(* Logix 5000 project; controller IF2_DEMO Emulate 5570 rev 20.12; software revision 20.04; part 3 of 8 *)
(* tags used below, declared in another part *)
   HMI_Motion : COUNTER;
   Next_Product : DINT;
   OEE_Part_Scrap_Old : DINT;
   OEE_Scrap_Labeler : DINT;
   OrderQty : DINT[4];
   PartCountRollOver : DINT;
   Product_Change : DINT;
   RefillLine : LineData;
   Timer1000ms : TIMER;
   Timer250ms : TIMER;
   WallClock : DINT[7];
   WC : WC[10];

PROGRAM FillerR   (* main routine MainRoutine *)
VAR
   Block_Delay : TIMER := (PRE := 15000);
   Blocked_L : BOOL;
   BottleNum : STRING;
   Ctrl_Bit : BOOL := 1;
   DownStream_Run : ALIAS FOR WC[3].EventTrigger[0].1;
   DownStream_Running : ALIAS FOR WC[3].EventTrigger[0].8;
   Events : Events := (DownTime.BreakdownCode := 6, Control.StandbyCode := 1, Control.Run := 1, Control.Auto := 1);
   Events_Control_Auto : ALIAS FOR WC_L.EventTrigger[0].5;
   Events_Control_OpStop : ALIAS FOR WC_L.EventTrigger[0].3;
   Events_Control_Run : ALIAS FOR WC_L.EventTrigger[0].1;
   Events_Control_Running : ALIAS FOR WC_L.EventTrigger[0].8;
   Events_Control_Standby : ALIAS FOR WC_L.EventTrigger[0].0;
   Events_Control_StandbyCode : ALIAS FOR WC_L.FlexREAL[1];
   Events_DownTime_Breakdown : ALIAS FOR WC_L.EventTrigger[0].2;
   Events_DownTime_BreakdownCode : ALIAS FOR WC_L.EventValue_REAL[2];
   Events_DownTime_Testing : ALIAS FOR WC_L.EventTrigger[0].7;
   Events_DownTime_UnschedMaint : ALIAS FOR WC_L.EventTrigger[0].6;
   Events_Operate_Load : ALIAS FOR WC_L.EventTrigger[0].10;
   Events_Operate_OrderProc : ALIAS FOR WC_L.EventTrigger[0].11;
   Events_Operate_Setup : ALIAS FOR WC_L.EventTrigger[0].9;
   FillOunces : INT;
   HMI : HMIVars := (ScrapRate := 5.0, SpeedControl := 100.0, PrevSpeed := 100.0, PartCountRollOver := 9999999, MfgTimeBase := 1, MaxEventDur := 14.0, MinEventDur := 5.0, EventsPerHr := 55, EventDur := 12.487433, RunDur := 51.79828, MinRunDur := 5.0);
   MfgOrders : MfgOrders := (CustomerName := 'Big-Mart', OrderName := 'BB21', OrderQty := 30000, ProdRate := 60.0, SetupTime := 37.0, PartName := 'STRAW-R40', WorkcellName := 'FillerR', OperationId := 17160304, PartNameSav := 'STRAW-R40');
   MfgOrders_CustomerName : ALIAS FOR WC_L.FlexSTRING[4];
   MfgOrders_OrderName : ALIAS FOR WC_L.FlexSTRING[3];
   MfgOrders_PartName : ALIAS FOR WC_L.FlexSTRING[0];
   Motion : DINT := 31;
   Motion_Counter : DINT := 2;
   Motion_Speed : DINT := 10;
   MotionCount : TIMER := (PRE := 900);
   OEE : OEE := (IdealCycleTime := 3.0);
   OEE_IdealCycleTime : ALIAS FOR WC_L.IdealCT;
   OEE_Parts_Good : ALIAS FOR WC_L.GoodParts;
   OEE_Parts_Scrap : ALIAS FOR WC_L.ScrapParts;
   OEE_Parts_Total : ALIAS FOR WC_L.TotalParts;
   onsbits : DINT;
   OperatorID : ALIAS FOR WC_L.FlexREAL[1];
   Pressure1 : ALIAS FOR WC_L.PV[0];   // PSI
   ProductColorCode : INT := 2;
   RecipeName : STRING;
   SIM : SimVars := (Run.PRE := 51798, Event.PRE := 5000, Setup.PRE := 5000, EventNumber := 11, UtilityBool[2] := 1);
        .UTILITYBOOL[2]   // First Scan Bit
   Starve_Delay : TIMER := (PRE := 15000);
   Starved_L : BOOL;
   StateValue : ALIAS FOR WC_L.MonitorValue[0];
   Suppress : Events;
   Temperature1 : ALIAS FOR WC_L.PV[1];   // DEG
   UpStream_Run : BOOL := 1;
   UpStream_Running : BOOL := 1;   // Not used-no upstream wc
   WC_L : ALIAS FOR WC[1];
END_VAR

ROUTINE MainRoutine   (* ladder *)
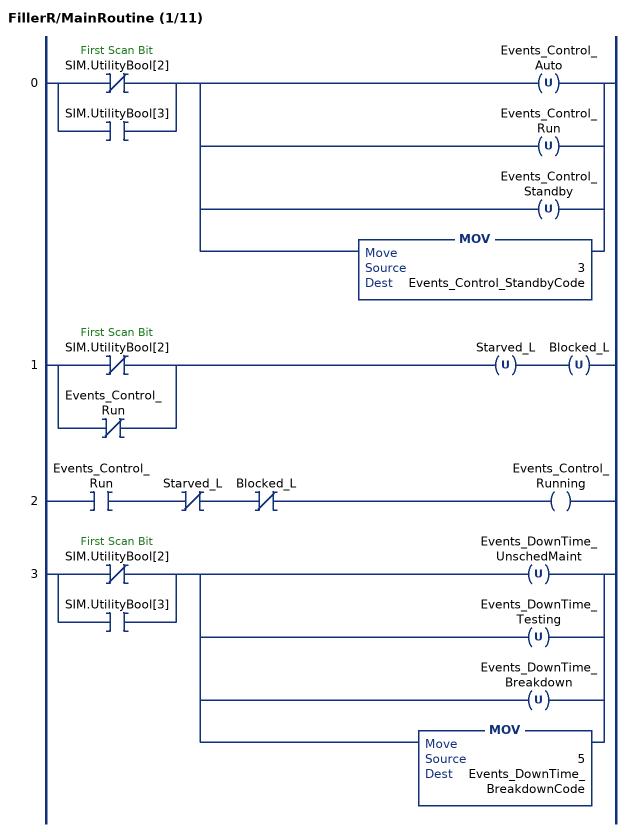
   0: [XIO(SIM.UtilityBool[2]) ,XIC(SIM.UtilityBool[3]) ][OTU(Events_Control_Auto) ,OTU(Events_Control_Run) ,OTU(Events_Control_Standby) ,MOV(3,Events_Control_StandbyCode) ];
   1: [XIO(SIM.UtilityBool[2]) ,XIO(Events_Control_Run) ]OTU(Starved_L)OTU(Blocked_L);
   2: XIC(Events_Control_Run)XIO(Starved_L)XIO(Blocked_L)OTE(Events_Control_Running);
   3: [XIO(SIM.UtilityBool[2]) ,XIC(SIM.UtilityBool[3]) ][OTU(Events_DownTime_UnschedMaint) ,OTU(Events_DownTime_Testing) ,OTU(Events_DownTime_Breakdown) ,MOV(5,Events_DownTime_BreakdownCode) ];
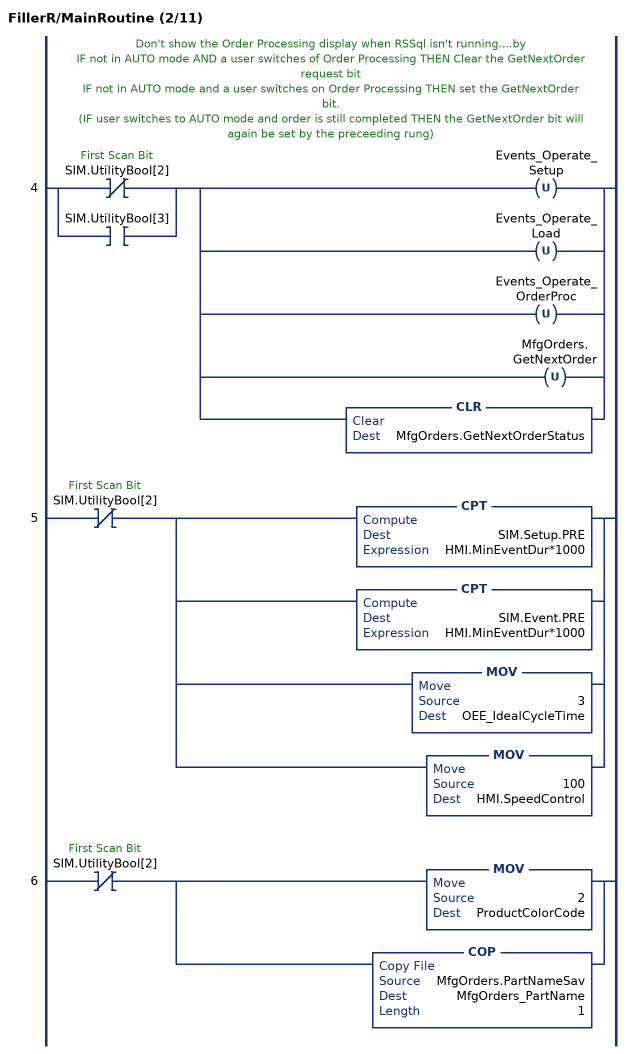
   // Don't show the Order Processing display when RSSql isn't running....by
   // IF not in AUTO mode AND a user switches of Order Processing THEN Clear the GetNextOrder request bit
   // IF not in AUTO mode and a user switches on Order Processing THEN set the GetNextOrder bit.
   // (IF user switches to AUTO mode and order is still completed THEN the GetNextOrder bit will again be set by the preceeding rung)
   4: [XIO(SIM.UtilityBool[2]) ,XIC(SIM.UtilityBool[3]) ][OTU(Events_Operate_Setup) ,OTU(Events_Operate_Load) ,OTU(Events_Operate_OrderProc) ,OTU(MfgOrders.GetNextOrder) ,CLR(MfgOrders.GetNextOrderStatus) ];
   5: XIO(SIM.UtilityBool[2])[CPT(SIM.Setup.PRE,HMI.MinEventDur*1000) ,CPT(SIM.Event.PRE,HMI.MinEventDur*1000) ,MOV(3,OEE_IdealCycleTime) ,MOV(100,HMI.SpeedControl) ];
   6: XIO(SIM.UtilityBool[2])[MOV(2,ProductColorCode) ,COP(MfgOrders.PartNameSav,MfgOrders_PartName,1) ];
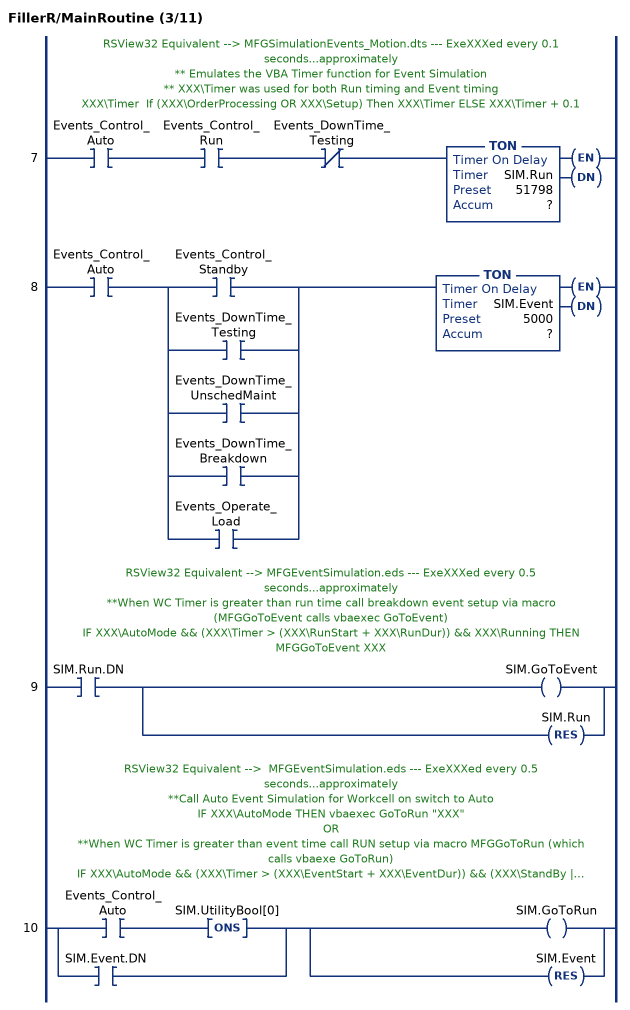
   // RSView32 Equivalent --> MFGSimulationEvents_Motion.dts --- ExeXXXed every 0.1 seconds...approximately
   // ** Emulates the VBA Timer function for Event Simulation
   // ** XXX\Timer was used for both Run timing and Event timing
   // XXX\Timer	If (XXX\OrderProcessing OR XXX\Setup) Then XXX\Timer ELSE XXX\Timer + 0.1
   7: XIC(Events_Control_Auto)XIC(Events_Control_Run)XIO(Events_DownTime_Testing)TON(SIM.Run,?,?);
   8: XIC(Events_Control_Auto)[XIC(Events_Control_Standby) ,XIC(Events_DownTime_Testing) ,XIC(Events_DownTime_UnschedMaint) ,XIC(Events_DownTime_Breakdown) ,XIC(Events_Operate_Load) ]TON(SIM.Event,?,?);
   // RSView32 Equivalent --> MFGEventSimulation.eds --- ExeXXXed every 0.5 seconds...approximately
   // **When WC Timer is greater than run time call breakdown event setup via macro (MFGGoToEvent calls vbaexec GoToEvent)
   // IF XXX\AutoMode && (XXX\Timer > (XXX\RunStart + XXX\RunDur)) && XXX\Running THEN MFGGoToEvent XXX
   9: XIC(SIM.Run.DN)[OTE(SIM.GoToEvent) ,RES(SIM.Run) ];
   // RSView32 Equivalent -->  MFGEventSimulation.eds --- ExeXXXed every 0.5 seconds...approximately
   // **Call Auto Event Simulation for Workcell on switch to Auto
   // IF XXX\AutoMode THEN vbaexec GoToRun "XXX"
   // OR
   // **When WC Timer is greater than event time call RUN setup via macro MFGGoToRun (which calls vbaexe GoToRun)
   // IF XXX\AutoMode && (XXX\Timer > (XXX\EventStart + XXX\EventDur)) && (XXX\StandBy || XXX\Test || XXX\UnSchedMaint || XXX\Breakdown ||XXX\Load) THEN MFGGoToRun XXX
   10: [XIC(Events_Control_Auto) ONS(SIM.UtilityBool[0]) ,XIC(SIM.Event.DN) ][OTE(SIM.GoToRun) ,RES(SIM.Event) ];
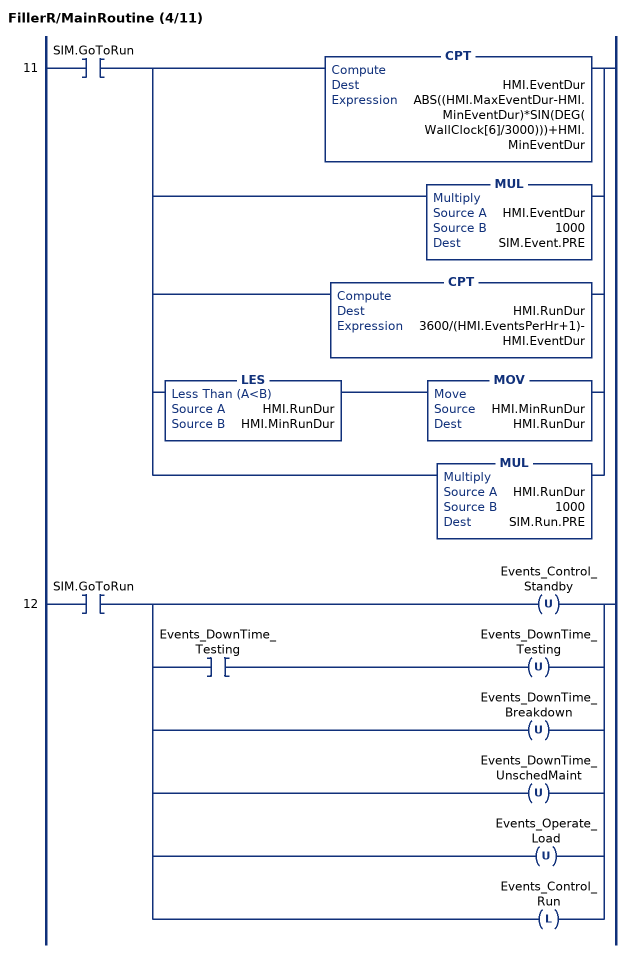
   11: XIC(SIM.GoToRun)[CPT(HMI.EventDur,ABS((HMI.MaxEventDur-HMI.MinEventDur)*SIN(DEG(WallClock[6]/3000)))+HMI.MinEventDur) ,MUL(HMI.EventDur,1000,SIM.Event.PRE) ,CPT(HMI.RunDur,3600/(HMI.EventsPerHr+1)-HMI.EventDur) ,LES(HMI.RunDur,HMI.MinRunDur) MOV(HMI.MinRunDur,HMI.RunDur) ,MUL(HMI.RunDur,1000,SIM.Run.PRE) ];
   12: XIC(SIM.GoToRun)[OTU(Events_Control_Standby) ,XIC(Events_DownTime_Testing) OTU(Events_DownTime_Testing) ,OTU(Events_DownTime_Breakdown) ,OTU(Events_DownTime_UnschedMaint) ,OTU(Events_Operate_Load) ,OTL(Events_Control_Run) ];
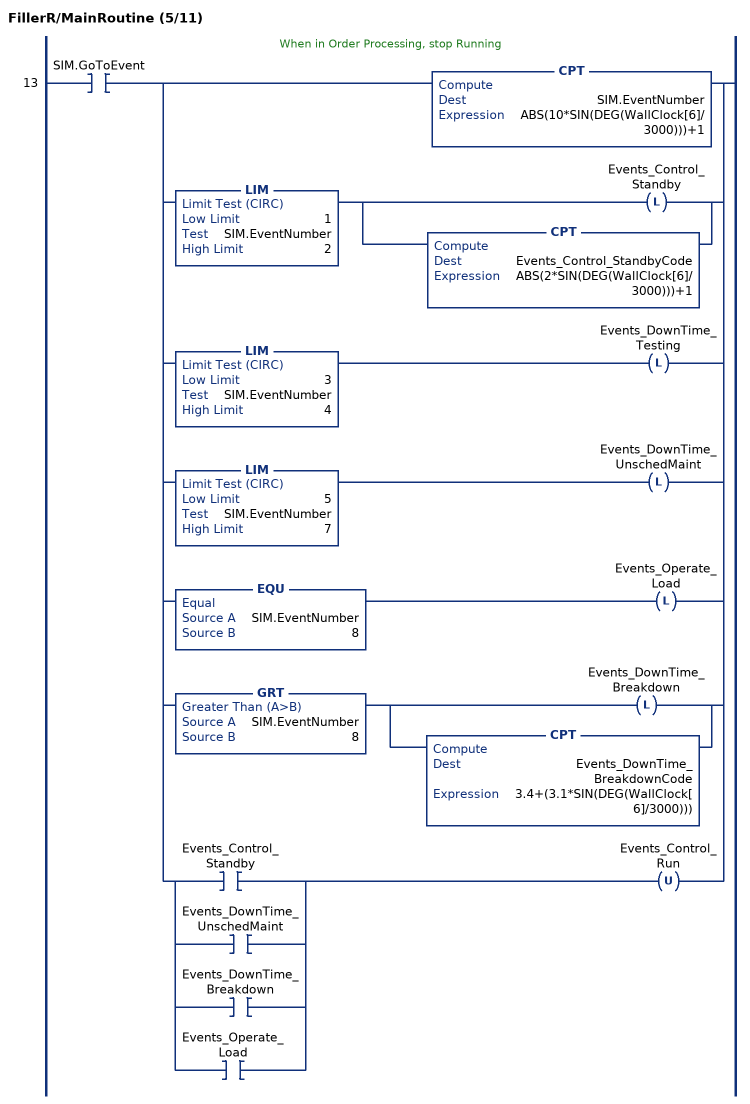
   // When in Order Processing, stop Running
   13: XIC(SIM.GoToEvent)[CPT(SIM.EventNumber,ABS(10*SIN(DEG(WallClock[6]/3000)))+1) ,LIM(1,SIM.EventNumber,2) [OTL(Events_Control_Standby) ,CPT(Events_Control_StandbyCode,ABS(2*SIN(DEG(WallClock[6]/3000)))+1) ] ,LIM(3,SIM.EventNumber,4) OTL(Events_DownTime_Testing) ,LIM(5,SIM.EventNumber,7) OTL(Events_DownTime_UnschedMaint) ,EQU(SIM.EventNumber,8) OTL(Events_Operate_Load) ,GRT(SIM.EventNumber,8) [OTL(Events_DownTime_Breakdown) ,CPT(Events_DownTime_BreakdownCode,3.4+(3.1*SIN(DEG(WallClock[6]/3000)))) ] ,[XIC(Events_Control_Standby) ,XIC(Events_DownTime_UnschedMaint) ,XIC(Events_DownTime_Breakdown) ,XIC(Events_Operate_Load) ] OTU(Events_Control_Run) ];
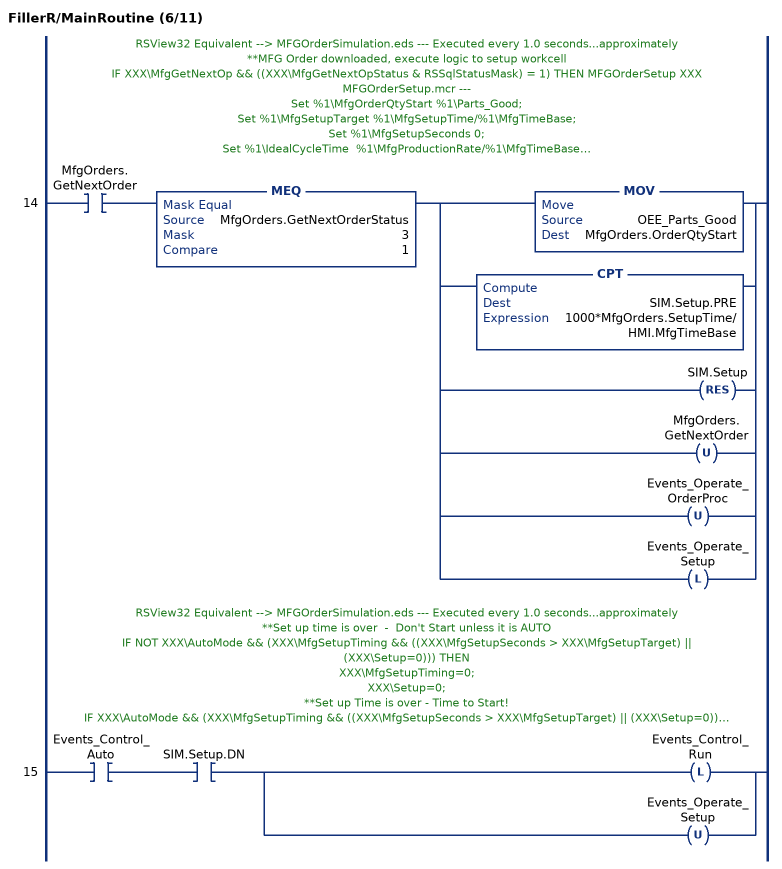
   // RSView32 Equivalent --> MFGOrderSimulation.eds --- Executed every 1.0 seconds...approximately
   // **MFG Order downloaded, execute logic to setup workcell
   // IF XXX\MfgGetNextOp && ((XXX\MfgGetNextOpStatus & RSSqlStatusMask) = 1) THEN MFGOrderSetup XXX
   // MFGOrderSetup.mcr ---
   // 	Set %1\MfgOrderQtyStart %1\Parts_Good;
   // 	Set %1\MfgSetupTarget %1\MfgSetupTime/%1\MfgTimeBase;
   // 	Set %1\MfgSetupSeconds 0;
   // 	Set %1\IdealCycleTime  %1\MfgProductionRate/%1\MfgTimeBase;
   // 	Set %1\MfgGetNextOp 0;
   // 	Set %1\Setup 1;
   // 	Set %1\OrderProcessing 0;
   // 	Set %1\MfgSetupTiming 1;
   14: XIC(MfgOrders.GetNextOrder)MEQ(MfgOrders.GetNextOrderStatus,3,1)[MOV(OEE_Parts_Good,MfgOrders.OrderQtyStart) ,CPT(SIM.Setup.PRE,1000*MfgOrders.SetupTime/HMI.MfgTimeBase) ,RES(SIM.Setup) ,OTU(MfgOrders.GetNextOrder) ,OTU(Events_Operate_OrderProc) ,OTL(Events_Operate_Setup) ];
   // RSView32 Equivalent --> MFGOrderSimulation.eds --- Executed every 1.0 seconds...approximately
   // **Set up time is over  -  Don't Start unless it is AUTO
   // IF NOT XXX\AutoMode && (XXX\MfgSetupTiming && ((XXX\MfgSetupSeconds > XXX\MfgSetupTarget) || (XXX\Setup=0))) THEN
   // 	XXX\MfgSetupTiming=0;
   // 	XXX\Setup=0;
   // **Set up Time is over - Time to Start!
   // IF XXX\AutoMode && (XXX\MfgSetupTiming && ((XXX\MfgSetupSeconds > XXX\MfgSetupTarget) || (XXX\Setup=0))) THEN
   // 	XXX\MfgSetupTiming=0;
   // 	XXX\Setup=0;
   // 	XXX\RUNNING=1
   15: XIC(Events_Control_Auto)XIC(SIM.Setup.DN)[OTL(Events_Control_Run) ,OTU(Events_Operate_Setup) ];
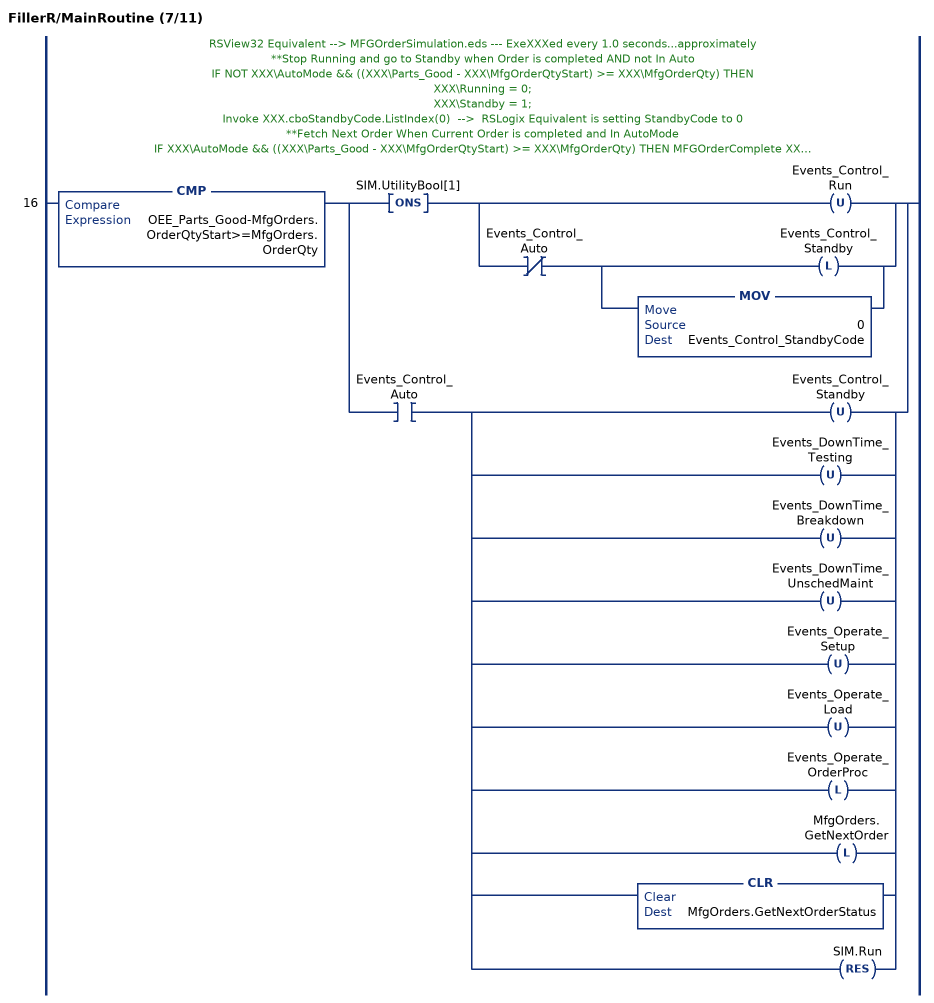
   // RSView32 Equivalent --> MFGOrderSimulation.eds --- ExeXXXed every 1.0 seconds...approximately
   // **Stop Running and go to Standby when Order is completed AND not In Auto
   // IF NOT XXX\AutoMode && ((XXX\Parts_Good - XXX\MfgOrderQtyStart) >= XXX\MfgOrderQty) THEN
   // 	XXX\Running = 0;
   // 	XXX\Standby = 1;
   // 	Invoke XXX.cboStandbyCode.ListIndex(0)  -->  RSLogix Equivalent is setting StandbyCode to 0
   // **Fetch Next Order When Current Order is completed and In AutoMode
   // IF XXX\AutoMode && ((XXX\Parts_Good - XXX\MfgOrderQtyStart) >= XXX\MfgOrderQty) THEN MFGOrderComplete XXX
   // MFGOrderComplete.mcr --- (Macros exeXXXed when called. %1 is the Workcell name -- typical all mcrs)
   // 	Set %1\RunStart %1\Timer;
   // 	Set %1\StandBy 0;
   // 	Set %1\Test 0;
   // 	Set %1\UnSchedMaint 0;
   // 	Set %1\Breakdown 0;
   // 	Set %1\Load 0;
   // 	Set %1\OrderProcessing 1;
   // 	Set %1\Running 0;
   // 	Set %1\MFGGetNextOpStatus 0;
   // 	Set %1\MFGGetNextOp 1
   16: CMP(OEE_Parts_Good-MfgOrders.OrderQtyStart>=MfgOrders.OrderQty)[ONS(SIM.UtilityBool[1]) [OTU(Events_Control_Run) ,XIO(Events_Control_Auto) [OTL(Events_Control_Standby) ,MOV(0,Events_Control_StandbyCode) ] ] ,XIC(Events_Control_Auto) [OTU(Events_Control_Standby) ,OTU(Events_DownTime_Testing) ,OTU(Events_DownTime_Breakdown) ,OTU(Events_DownTime_UnschedMaint) ,OTU(Events_Operate_Setup) ,OTU(Events_Operate_Load) ,OTL(Events_Operate_OrderProc) ,OTL(MfgOrders.GetNextOrder) ,CLR(MfgOrders.GetNextOrderStatus) ,RES(SIM.Run) ] ];
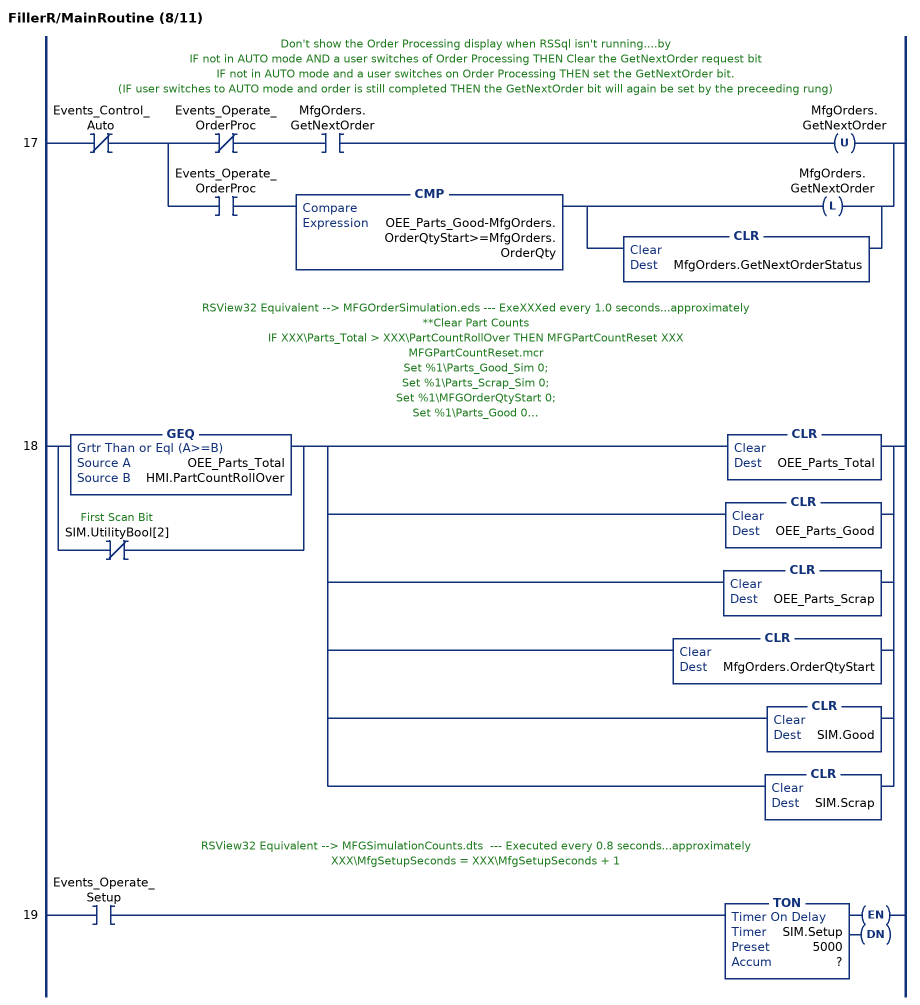
   // Don't show the Order Processing display when RSSql isn't running....by
   // IF not in AUTO mode AND a user switches of Order Processing THEN Clear the GetNextOrder request bit
   // IF not in AUTO mode and a user switches on Order Processing THEN set the GetNextOrder bit.
   // (IF user switches to AUTO mode and order is still completed THEN the GetNextOrder bit will again be set by the preceeding rung)
   17: XIO(Events_Control_Auto)[XIO(Events_Operate_OrderProc) XIC(MfgOrders.GetNextOrder) OTU(MfgOrders.GetNextOrder) ,XIC(Events_Operate_OrderProc) CMP(OEE_Parts_Good-MfgOrders.OrderQtyStart>=MfgOrders.OrderQty) [OTL(MfgOrders.GetNextOrder) ,CLR(MfgOrders.GetNextOrderStatus) ] ];
   // RSView32 Equivalent --> MFGOrderSimulation.eds --- ExeXXXed every 1.0 seconds...approximately
   // **Clear Part Counts
   // IF XXX\Parts_Total > XXX\PartCountRollOver THEN MFGPartCountReset XXX
   // MFGPartCountReset.mcr
   // 	Set %1\Parts_Good_Sim 0;
   // 	Set %1\Parts_Scrap_Sim 0;
   // 	Set %1\MFGOrderQtyStart 0;
   // 	Set %1\Parts_Good 0;
   // 	Set %1\Parts_Scrap 0;
   // 	Set %1\Parts_Total 0
   18: [GEQ(OEE_Parts_Total,HMI.PartCountRollOver) ,XIO(SIM.UtilityBool[2]) ][CLR(OEE_Parts_Total) ,CLR(OEE_Parts_Good) ,CLR(OEE_Parts_Scrap) ,CLR(MfgOrders.OrderQtyStart) ,CLR(SIM.Good) ,CLR(SIM.Scrap) ];
   // RSView32 Equivalent --> MFGSimulationCounts.dts	--- Executed every 0.8 seconds...approximately
   // XXX\MfgSetupSeconds = XXX\MfgSetupSeconds + 1
   19: XIC(Events_Operate_Setup)TON(SIM.Setup,?,?);
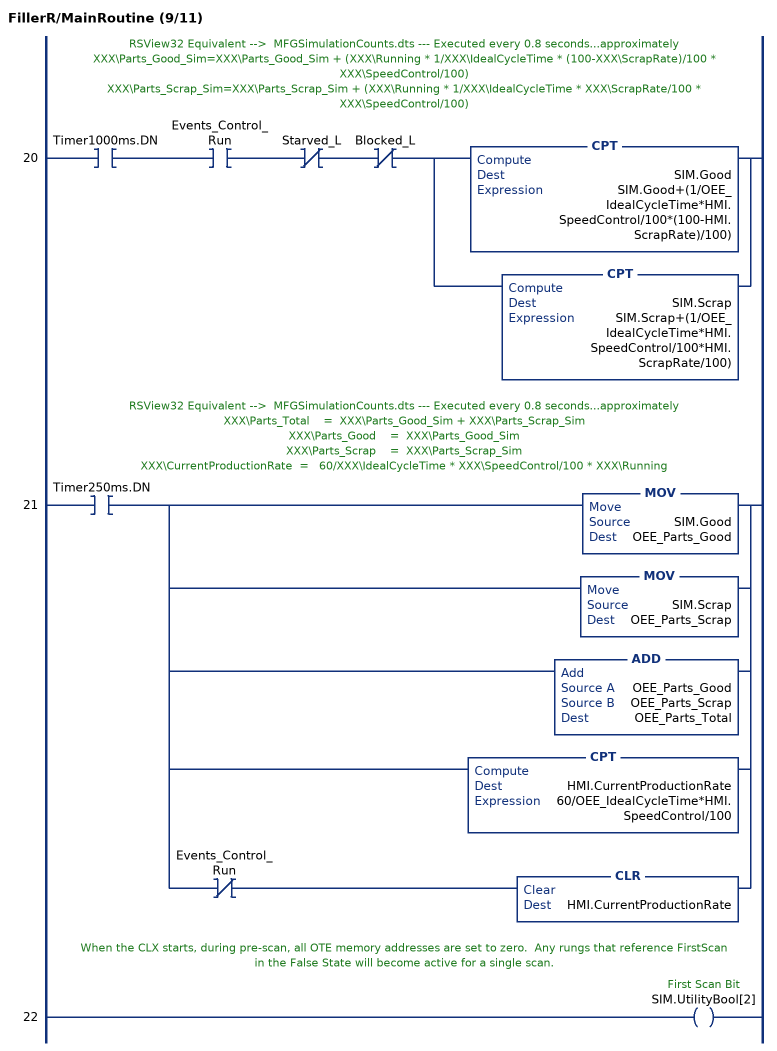
   // RSView32 Equivalent -->  MFGSimulationCounts.dts --- Executed every 0.8 seconds...approximately
   // XXX\Parts_Good_Sim=XXX\Parts_Good_Sim + (XXX\Running * 1/XXX\IdealCycleTime * (100-XXX\ScrapRate)/100 * XXX\SpeedControl/100)
   // XXX\Parts_Scrap_Sim=XXX\Parts_Scrap_Sim + (XXX\Running * 1/XXX\IdealCycleTime * XXX\ScrapRate/100 * XXX\SpeedControl/100)
   20: XIC(Timer1000ms.DN)XIC(Events_Control_Run)XIO(Starved_L)XIO(Blocked_L)[CPT(SIM.Good,SIM.Good+(1/OEE_IdealCycleTime*HMI.SpeedControl/100*(100-HMI.ScrapRate)/100)) ,CPT(SIM.Scrap,SIM.Scrap+(1/OEE_IdealCycleTime*HMI.SpeedControl/100*HMI.ScrapRate/100)) ];
   // RSView32 Equivalent -->  MFGSimulationCounts.dts --- Executed every 0.8 seconds...approximately
   // XXX\Parts_Total		=	XXX\Parts_Good_Sim + XXX\Parts_Scrap_Sim
   // XXX\Parts_Good		=	XXX\Parts_Good_Sim
   // XXX\Parts_Scrap		=	XXX\Parts_Scrap_Sim
   // XXX\CurrentProductionRate  = 	60/XXX\IdealCycleTime * XXX\SpeedControl/100 * XXX\Running
   21: XIC(Timer250ms.DN)[[MOV(SIM.Good,OEE_Parts_Good) ,MOV(SIM.Scrap,OEE_Parts_Scrap) ,ADD(OEE_Parts_Good,OEE_Parts_Scrap,OEE_Parts_Total) ] ,CPT(HMI.CurrentProductionRate,60/OEE_IdealCycleTime*HMI.SpeedControl/100) ,XIO(Events_Control_Run) CLR(HMI.CurrentProductionRate) ];
   // When the CLX starts, during pre-scan, all OTE memory addresses are set to zero.  Any rungs that reference FirstScan in the False State will become active for a single scan.
   22: OTE(SIM.UtilityBool[2]);
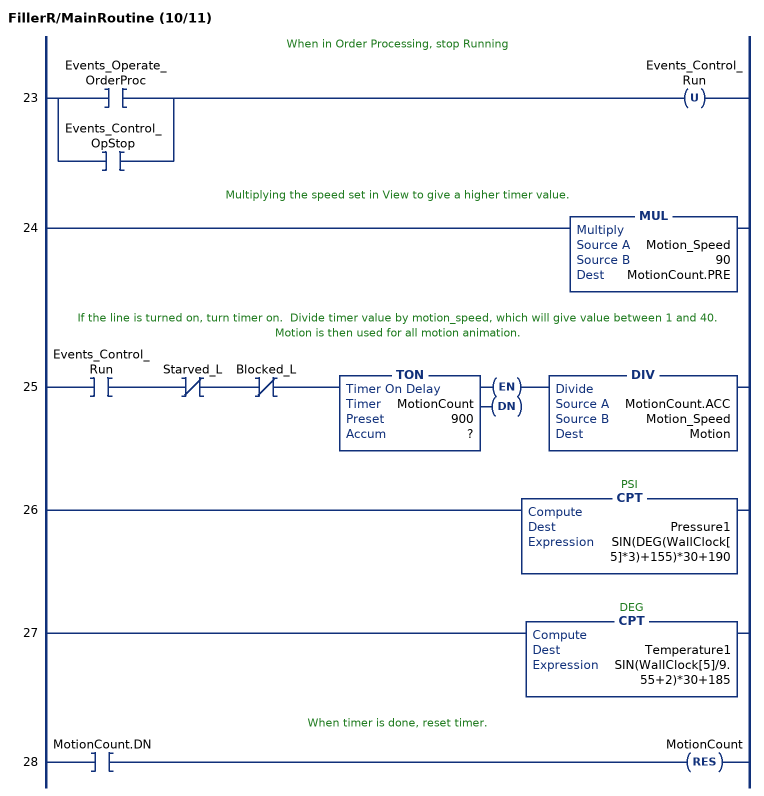
   // When in Order Processing, stop Running
   23: [XIC(Events_Operate_OrderProc) ,XIC(Events_Control_OpStop) ]OTU(Events_Control_Run);
   // Multiplying the speed set in View to give a higher timer value.
   24: MUL(Motion_Speed,90,MotionCount.PRE);
   // If the line is turned on, turn timer on.  Divide timer value by motion_speed, which will give value between 1 and 40.  Motion is then used for all motion animation.
   25: XIC(Events_Control_Run)XIO(Starved_L)XIO(Blocked_L)TON(MotionCount,?,?)DIV(MotionCount.ACC,Motion_Speed,Motion);
   26: CPT(Pressure1,SIN(DEG(WallClock[5]*3)+155)*30+190);
   27: CPT(Temperature1,SIN(WallClock[5]/9.55+2)*30+185);
   // When timer is done, reset timer.
   28: XIC(MotionCount.DN)RES(MotionCount);
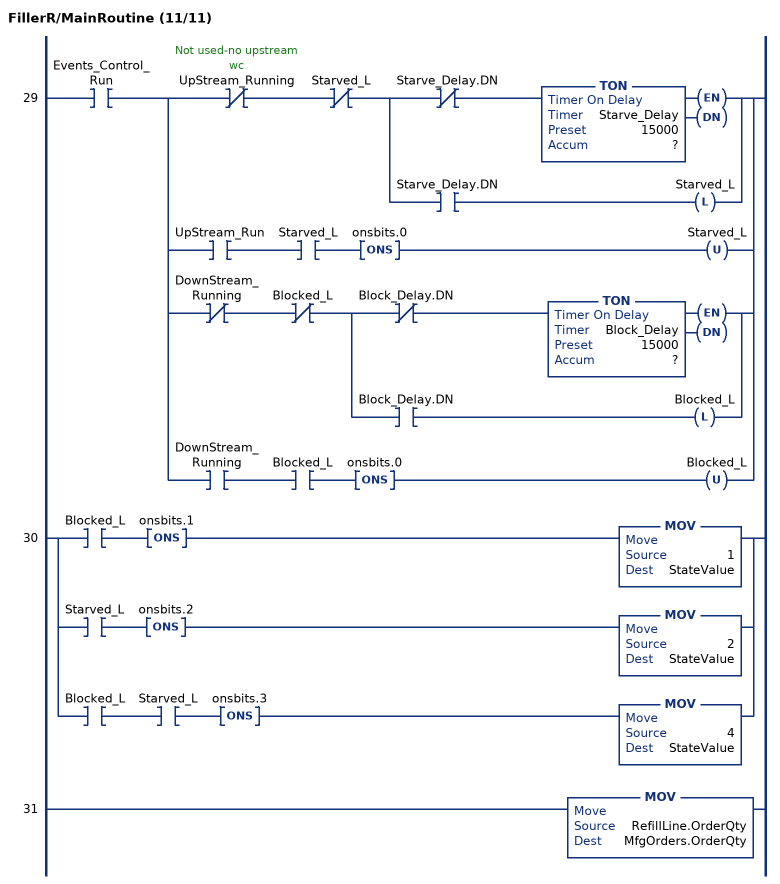
   29: XIC(Events_Control_Run)[[XIO(UpStream_Running) XIO(Starved_L) [XIO(Starve_Delay.DN) TON(Starve_Delay,?,?) ,XIC(Starve_Delay.DN) OTL(Starved_L) ] ,XIC(UpStream_Run) XIC(Starved_L) ONS(onsbits.0) OTU(Starved_L) ] ,[XIO(DownStream_Running) XIO(Blocked_L) [XIO(Block_Delay.DN) TON(Block_Delay,?,?) ,XIC(Block_Delay.DN) OTL(Blocked_L) ] ,XIC(DownStream_Running) XIC(Blocked_L) ONS(onsbits.0) OTU(Blocked_L) ] ];
   30: [XIC(Blocked_L) ONS(onsbits.1) MOV(1,StateValue) ,XIC(Starved_L) ONS(onsbits.2) MOV(2,StateValue) ,XIC(Blocked_L) XIC(Starved_L) ONS(onsbits.3) MOV(4,StateValue) ];
   31: MOV(RefillLine.OrderQty,MfgOrders.OrderQty);
END_ROUTINE
END_PROGRAM

PROGRAM LabelerD   (* main routine MainRoutine *)
VAR
   Alarm_Labeler1_Blocked : ALARM_DIGITAL;
   Alarm_Labeler1_Breakdown : ALARM_DIGITAL;
   Alarm_Labeler1_Starved : ALARM_DIGITAL;
   Alarm_Labeler1_Stopped : ALARM_DIGITAL;
   Block_Delay : TIMER := (PRE := 15000);
   Blocked_Condition : BOOL;
   Blocked_L : BOOL;
   BottleNum : STRING;
   Breakdown_Event_ONS : BOOL := 1;
   Breakdown_Labeler_Simulation : TIMER := (PRE := 300000, ACC := 53438, EN := 1, TT := 1);
   Breakdown_Labeler_Simulator_Down_Switch : BOOL;
   Breakdown_Occurance_Time : DINT := 260000;
   Breakdown_Variation_Stepper : DINT := 2;
   Ctrl_Bit : BOOL;
   DownStream_Run : ALIAS FOR WC[8].EventTrigger[0].1;
   DownStream_Running : ALIAS FOR WC[8].EventTrigger[0].8;
   Events : Events := (DownTime.BreakdownCode := 5, Control.StandbyCode := 1, Control.Run := 1, Control.Auto := 1);
   Events_Control_Auto : ALIAS FOR WC_L.EventTrigger[0].5;
   Events_Control_OpStop : ALIAS FOR WC_L.EventTrigger[0].3;
   Events_Control_Run : ALIAS FOR WC_L.EventTrigger[0].1;
   Events_Control_Running : ALIAS FOR WC_L.EventTrigger[0].8;
   Events_Control_Standby : ALIAS FOR WC_L.EventTrigger[0].0;
   Events_Control_StandbyCode : ALIAS FOR WC_L.EventValue_REAL[1];
   Events_DownTime_Breakdown : ALIAS FOR WC_L.EventTrigger[0].2;
   Events_DownTime_BreakdownCode : ALIAS FOR WC_L.EventValue_REAL[2];
   Events_DownTime_Testing : ALIAS FOR WC_L.EventTrigger[0].7;
   Events_DownTime_UnschedMaint : ALIAS FOR WC_L.EventTrigger[0].6;
   Events_Operate_Load : ALIAS FOR WC_L.EventTrigger[0].10;
   Events_Operate_OrderProc : ALIAS FOR WC_L.EventTrigger[0].11;
   Events_Operate_Setup : ALIAS FOR WC_L.EventTrigger[0].9;
   Expected_Full_Production_Rate : DINT := 113;
   FillOunces : INT;
   HMI : HMIVars := (ScrapRate := 6.0, SpeedControl := 400.0, PrevSpeed := 400.0, CurrentProductionRate := 120.0, PartCountRollOver := 99999999, MfgTimeBase := 1, MaxEventDur := 12.0, MinEventDur := 4.0, EventsPerHr := 50, EventDur := 4.99532, RunDur := 65.59291, MinRunDur := 5.0);
   Labeler : FTVPDemoWorkCell := (RunState := 1, Temperature := 105, GoodParts := 2066, ScrapParts := 924, ScrapRate := 9, ProductionRate := 119, Pressure := 143, OrderName := 'GF-08-CZ-525', CustomerName := 'Soda Inc.', PartName := 'GF-11');
   Labeler_Bottler_Per_Min : DINT := 113;
   Labeler_Start : BOOL := 1;
   Labeler_State : DINT;
   Labeler_Status : DINT := 1;
   Labeler_Stop : BOOL;
   MfgOrders : MfgOrders := (CustomerName := 'Big-Mart', OrderName := 'C321', ProdRate := 60.0, PartName := 'Apple-D12', WorkcellName := 'LabelerD', PartNameSav := 'Apple-D12');
   MfgOrders_CustomerName : ALIAS FOR WC_L.FlexSTRING[4];
   MfgOrders_OrderName : ALIAS FOR WC_L.FlexSTRING[3];
   MfgOrders_PartName : ALIAS FOR WC_L.FlexSTRING[0];
   Motion : DINT := 55;
   Motion_Counter : DINT;
   Motion_Speed : DINT := 9;
   MotionAnimation : TIMER := (PRE := 5000, ACC := 3164, EN := 1, TT := 1);
   MotionCount : TIMER := (PRE := 810, ACC := 501, EN := 1, TT := 1);
   OEE : OEE := (IdealCycleTime := 2.0);
   OEE_Availability : REAL;
   OEE_IdealCycleTime : ALIAS FOR WC_L.IdealCT;
   OEE_Overall : REAL;
   OEE_Parts_Good : ALIAS FOR WC_L.GoodParts;
   OEE_Parts_Scrap : ALIAS FOR WC_L.ScrapParts;
   OEE_Parts_Total : ALIAS FOR WC_L.TotalParts;
   OEE_Performance : REAL;
   OEE_Quality : REAL := 0.8826568;
   onsbits : DINT;
   OperatorID : ALIAS FOR WC_L.FlexREAL[1];
   Pressure1 : ALIAS FOR WC_L.PV[0];   // PSI
   ProductColor : DINT := 1;
   ProductColorCode : INT := 3;
   RecipeName : STRING;
   SIM : SimVars := (Run.PRE := 65593, Event.PRE := 4000, Setup.PRE := 4000, Good := 1403.0316, Scrap := 186.5234, EventNumber := 9, UtilityBool[1] := 1, UtilityBool[2] := 1);
        .UTILITYBOOL[0]   // Enter Auto Mode ONS
        .UTILITYBOOL[1]   // Work Order Complete ONS
        .UTILITYBOOL[2]   // First Scan Bit
   Starve_Block_Labeler_ONS : BOOL;
   Starve_Delay : TIMER := (PRE := 15000);
   Starved_Condition : BOOL;
   Starved_L : BOOL;
   StateValue : ALIAS FOR WC_L.MonitorValue[0];
   Suppress : Events;
   Temperature1 : ALIAS FOR WC_L.PV[1];   // DEG
   TempReadTrigger : TIMER := (PRE := 5000, ACC := 3687, EN := 1, TT := 1);
   TempTimer : TIMER := (PRE := 10000, ACC := 3665, EN := 1, TT := 1);
   TempTimer2 : TIMER := (PRE := 5000, ACC := 3687, EN := 1, TT := 1);
   Timer_To_Labeler_Changeover : TIMER := (PRE := 30000);
   UpStream_Run : ALIAS FOR WC[2].EventTrigger[0].1;
   UpStream_Running : ALIAS FOR WC[2].EventTrigger[0].8;
   WC_L : ALIAS FOR WC[4];
END_VAR

ROUTINE MainRoutine   (* ladder *)
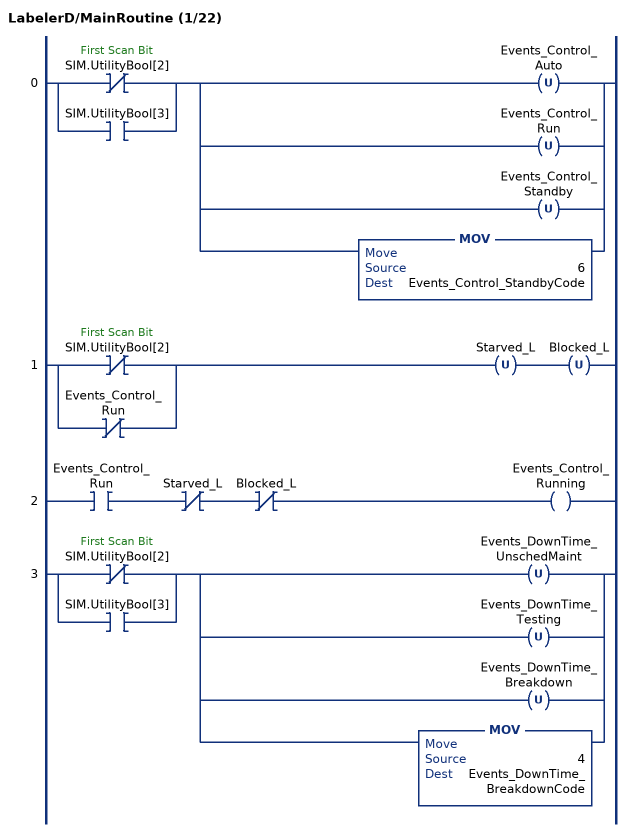
   0: [XIO(SIM.UtilityBool[2]) ,XIC(SIM.UtilityBool[3]) ][OTU(Events_Control_Auto) ,OTU(Events_Control_Run) ,OTU(Events_Control_Standby) ,MOV(6,Events_Control_StandbyCode) ];
   1: [XIO(SIM.UtilityBool[2]) ,XIO(Events_Control_Run) ]OTU(Starved_L)OTU(Blocked_L);
   2: XIC(Events_Control_Run)XIO(Starved_L)XIO(Blocked_L)OTE(Events_Control_Running);
   3: [XIO(SIM.UtilityBool[2]) ,XIC(SIM.UtilityBool[3]) ][OTU(Events_DownTime_UnschedMaint) ,OTU(Events_DownTime_Testing) ,OTU(Events_DownTime_Breakdown) ,MOV(4,Events_DownTime_BreakdownCode) ];
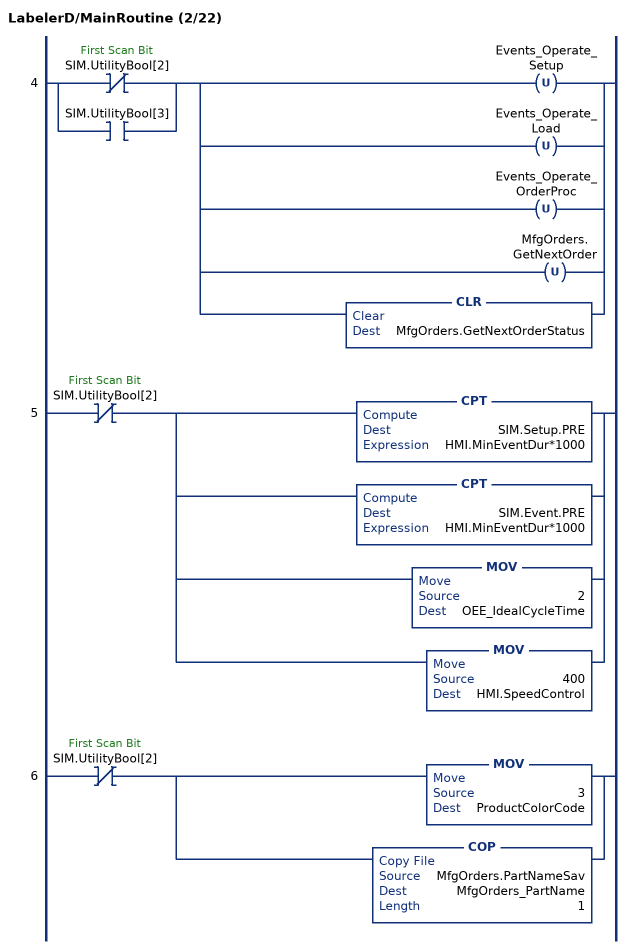
   4: [XIO(SIM.UtilityBool[2]) ,XIC(SIM.UtilityBool[3]) ][OTU(Events_Operate_Setup) ,OTU(Events_Operate_Load) ,OTU(Events_Operate_OrderProc) ,OTU(MfgOrders.GetNextOrder) ,CLR(MfgOrders.GetNextOrderStatus) ];
   5: XIO(SIM.UtilityBool[2])[CPT(SIM.Setup.PRE,HMI.MinEventDur*1000) ,CPT(SIM.Event.PRE,HMI.MinEventDur*1000) ,MOV(2,OEE_IdealCycleTime) ,MOV(400,HMI.SpeedControl) ];
   6: XIO(SIM.UtilityBool[2])[MOV(3,ProductColorCode) ,COP(MfgOrders.PartNameSav,MfgOrders_PartName,1) ];
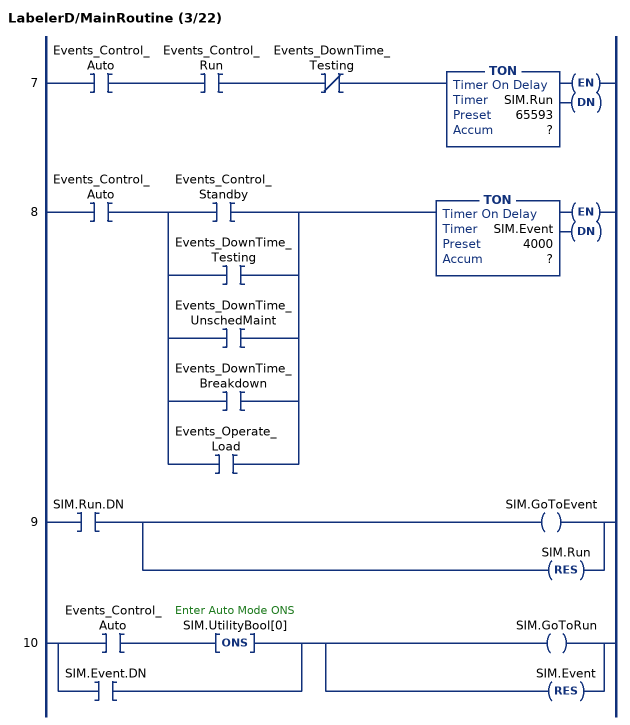
   7: XIC(Events_Control_Auto)XIC(Events_Control_Run)XIO(Events_DownTime_Testing)TON(SIM.Run,?,?);
   8: XIC(Events_Control_Auto)[XIC(Events_Control_Standby) ,XIC(Events_DownTime_Testing) ,XIC(Events_DownTime_UnschedMaint) ,XIC(Events_DownTime_Breakdown) ,XIC(Events_Operate_Load) ]TON(SIM.Event,?,?);
   9: XIC(SIM.Run.DN)[OTE(SIM.GoToEvent) ,RES(SIM.Run) ];
   10: [XIC(Events_Control_Auto) ONS(SIM.UtilityBool[0]) ,XIC(SIM.Event.DN) ][OTE(SIM.GoToRun) ,RES(SIM.Event) ];
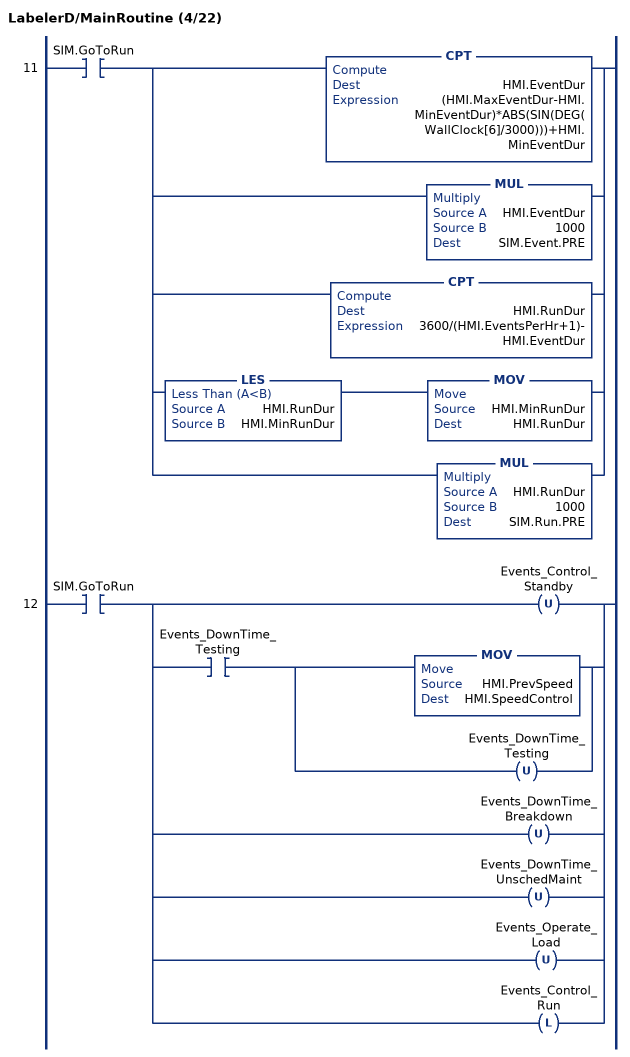
   11: XIC(SIM.GoToRun)[CPT(HMI.EventDur,(HMI.MaxEventDur-HMI.MinEventDur)*ABS(SIN(DEG(WallClock[6]/3000)))+HMI.MinEventDur) ,MUL(HMI.EventDur,1000,SIM.Event.PRE) ,CPT(HMI.RunDur,3600/(HMI.EventsPerHr+1)-HMI.EventDur) ,LES(HMI.RunDur,HMI.MinRunDur) MOV(HMI.MinRunDur,HMI.RunDur) ,MUL(HMI.RunDur,1000,SIM.Run.PRE) ];
   12: XIC(SIM.GoToRun)[OTU(Events_Control_Standby) ,XIC(Events_DownTime_Testing) [MOV(HMI.PrevSpeed,HMI.SpeedControl) ,OTU(Events_DownTime_Testing) ] ,OTU(Events_DownTime_Breakdown) ,OTU(Events_DownTime_UnschedMaint) ,OTU(Events_Operate_Load) ,OTL(Events_Control_Run) ];
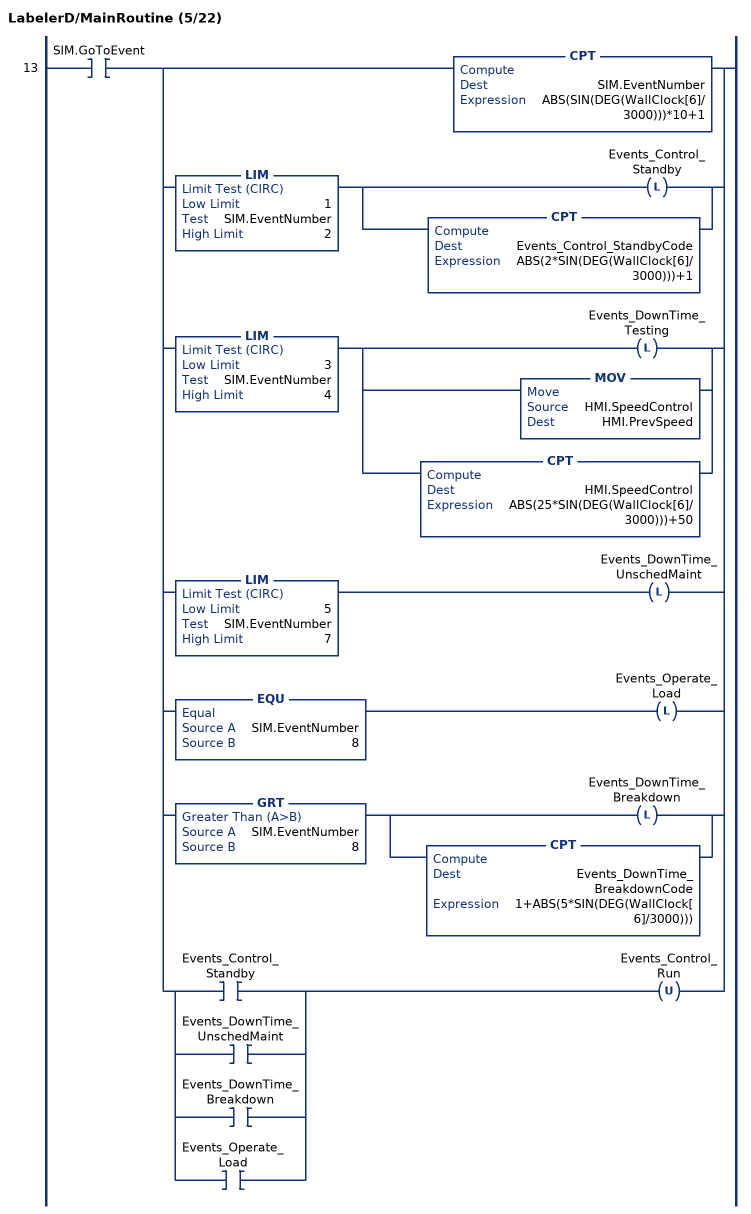
   13: XIC(SIM.GoToEvent)[CPT(SIM.EventNumber,ABS(SIN(DEG(WallClock[6]/3000)))*10+1) ,LIM(1,SIM.EventNumber,2) [OTL(Events_Control_Standby) ,CPT(Events_Control_StandbyCode,ABS(2*SIN(DEG(WallClock[6]/3000)))+1) ] ,LIM(3,SIM.EventNumber,4) [OTL(Events_DownTime_Testing) ,MOV(HMI.SpeedControl,HMI.PrevSpeed) ,CPT(HMI.SpeedControl,ABS(25*SIN(DEG(WallClock[6]/3000)))+50) ] ,LIM(5,SIM.EventNumber,7) OTL(Events_DownTime_UnschedMaint) ,EQU(SIM.EventNumber,8) OTL(Events_Operate_Load) ,GRT(SIM.EventNumber,8) [OTL(Events_DownTime_Breakdown) ,CPT(Events_DownTime_BreakdownCode,1+ABS(5*SIN(DEG(WallClock[6]/3000)))) ] ,[XIC(Events_Control_Standby) ,XIC(Events_DownTime_UnschedMaint) ,XIC(Events_DownTime_Breakdown) ,XIC(Events_Operate_Load) ] OTU(Events_Control_Run) ];
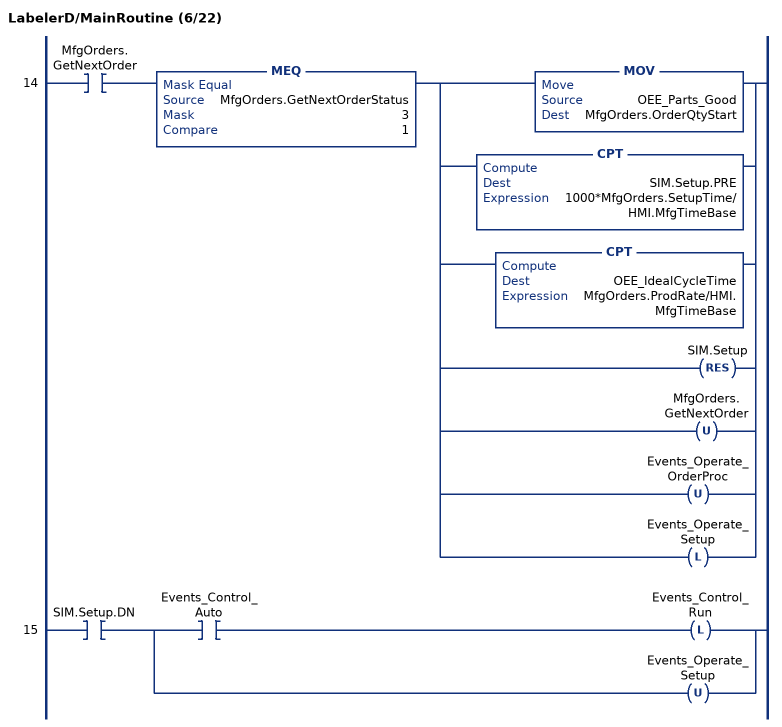
   14: XIC(MfgOrders.GetNextOrder)MEQ(MfgOrders.GetNextOrderStatus,3,1)[MOV(OEE_Parts_Good,MfgOrders.OrderQtyStart) ,CPT(SIM.Setup.PRE,1000*MfgOrders.SetupTime/HMI.MfgTimeBase) ,CPT(OEE_IdealCycleTime,MfgOrders.ProdRate/HMI.MfgTimeBase) ,RES(SIM.Setup) ,OTU(MfgOrders.GetNextOrder) ,OTU(Events_Operate_OrderProc) ,OTL(Events_Operate_Setup) ];
   15: XIC(SIM.Setup.DN)[XIC(Events_Control_Auto) OTL(Events_Control_Run) ,OTU(Events_Operate_Setup) ];
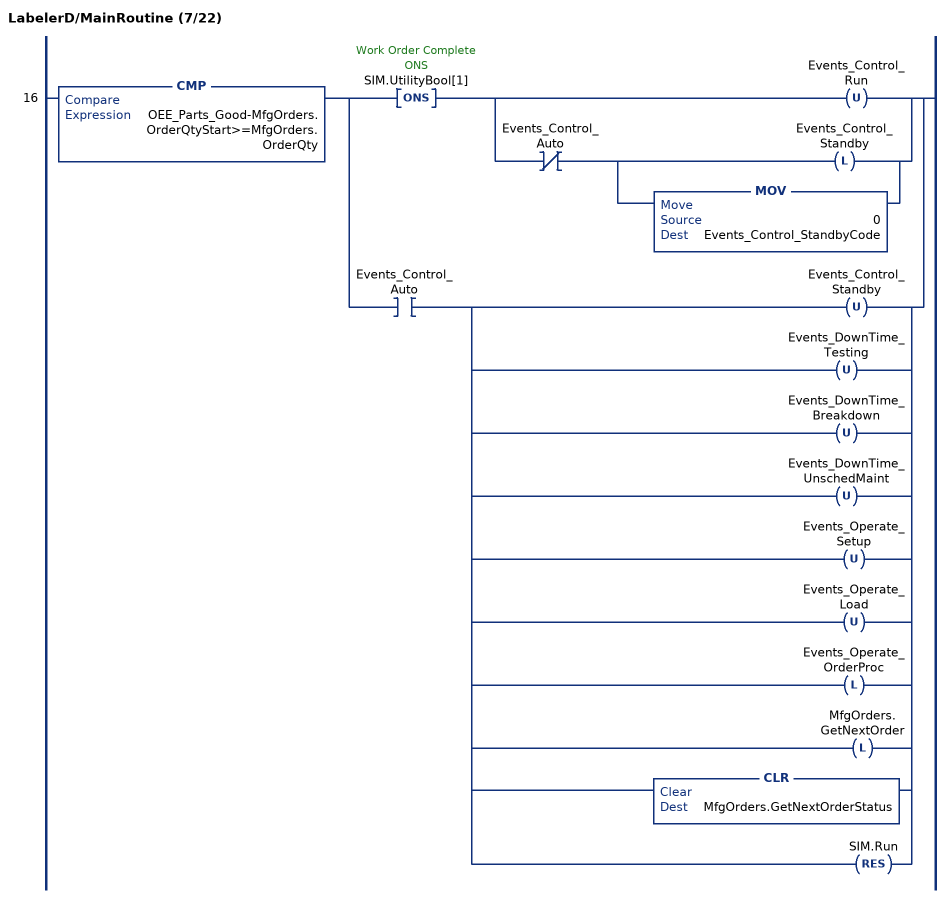
   16: CMP(OEE_Parts_Good-MfgOrders.OrderQtyStart>=MfgOrders.OrderQty)[ONS(SIM.UtilityBool[1]) [OTU(Events_Control_Run) ,XIO(Events_Control_Auto) [OTL(Events_Control_Standby) ,MOV(0,Events_Control_StandbyCode) ] ] ,XIC(Events_Control_Auto) [OTU(Events_Control_Standby) ,OTU(Events_DownTime_Testing) ,OTU(Events_DownTime_Breakdown) ,OTU(Events_DownTime_UnschedMaint) ,OTU(Events_Operate_Setup) ,OTU(Events_Operate_Load) ,OTL(Events_Operate_OrderProc) ,OTL(MfgOrders.GetNextOrder) ,CLR(MfgOrders.GetNextOrderStatus) ,RES(SIM.Run) ] ];
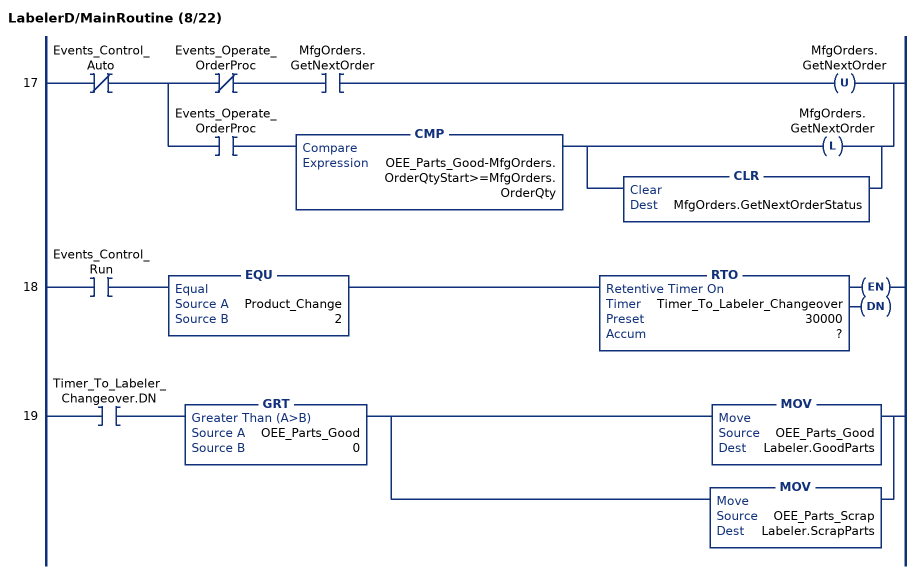
   17: XIO(Events_Control_Auto)[XIO(Events_Operate_OrderProc) XIC(MfgOrders.GetNextOrder) OTU(MfgOrders.GetNextOrder) ,XIC(Events_Operate_OrderProc) CMP(OEE_Parts_Good-MfgOrders.OrderQtyStart>=MfgOrders.OrderQty) [OTL(MfgOrders.GetNextOrder) ,CLR(MfgOrders.GetNextOrderStatus) ] ];
   18: XIC(Events_Control_Run)EQU(Product_Change,2)RTO(Timer_To_Labeler_Changeover,?,?);
   19: XIC(Timer_To_Labeler_Changeover.DN)GRT(OEE_Parts_Good,0)[MOV(OEE_Parts_Good,Labeler.GoodParts) ,MOV(OEE_Parts_Scrap,Labeler.ScrapParts) ];
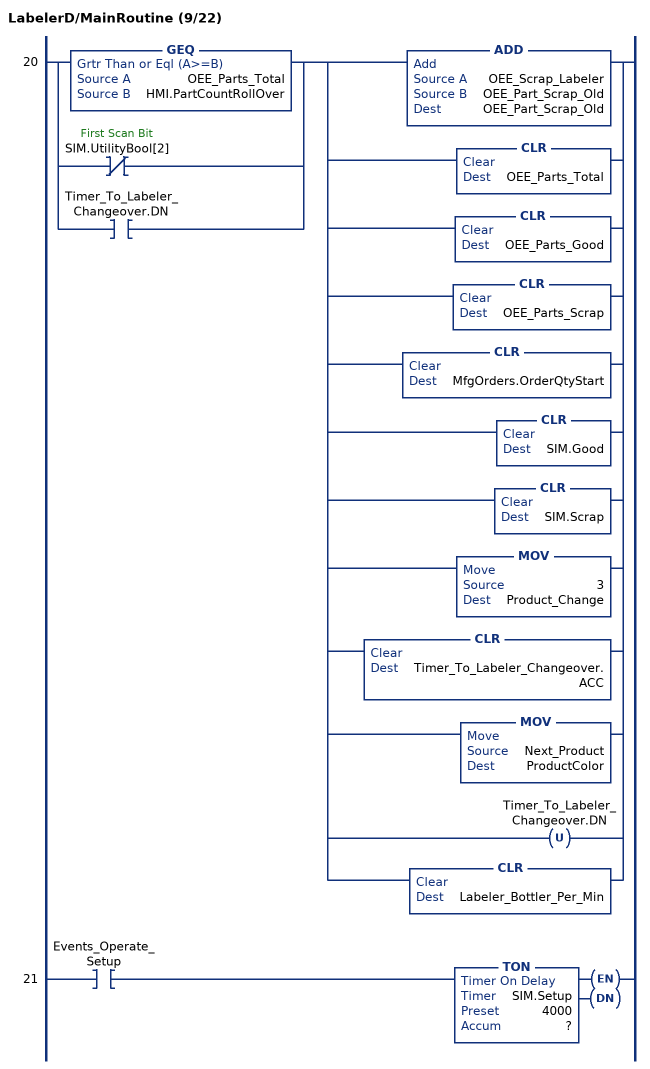
   20: [GEQ(OEE_Parts_Total,HMI.PartCountRollOver) ,XIO(SIM.UtilityBool[2]) ,XIC(Timer_To_Labeler_Changeover.DN) ][ADD(OEE_Scrap_Labeler,OEE_Part_Scrap_Old,OEE_Part_Scrap_Old) ,CLR(OEE_Parts_Total) ,CLR(OEE_Parts_Good) ,CLR(OEE_Parts_Scrap) ,CLR(MfgOrders.OrderQtyStart) ,CLR(SIM.Good) ,CLR(SIM.Scrap) ,MOV(3,Product_Change) ,CLR(Timer_To_Labeler_Changeover.ACC) ,MOV(Next_Product,ProductColor) ,OTU(Timer_To_Labeler_Changeover.DN) ,CLR(Labeler_Bottler_Per_Min) ];
   21: XIC(Events_Operate_Setup)TON(SIM.Setup,?,?);
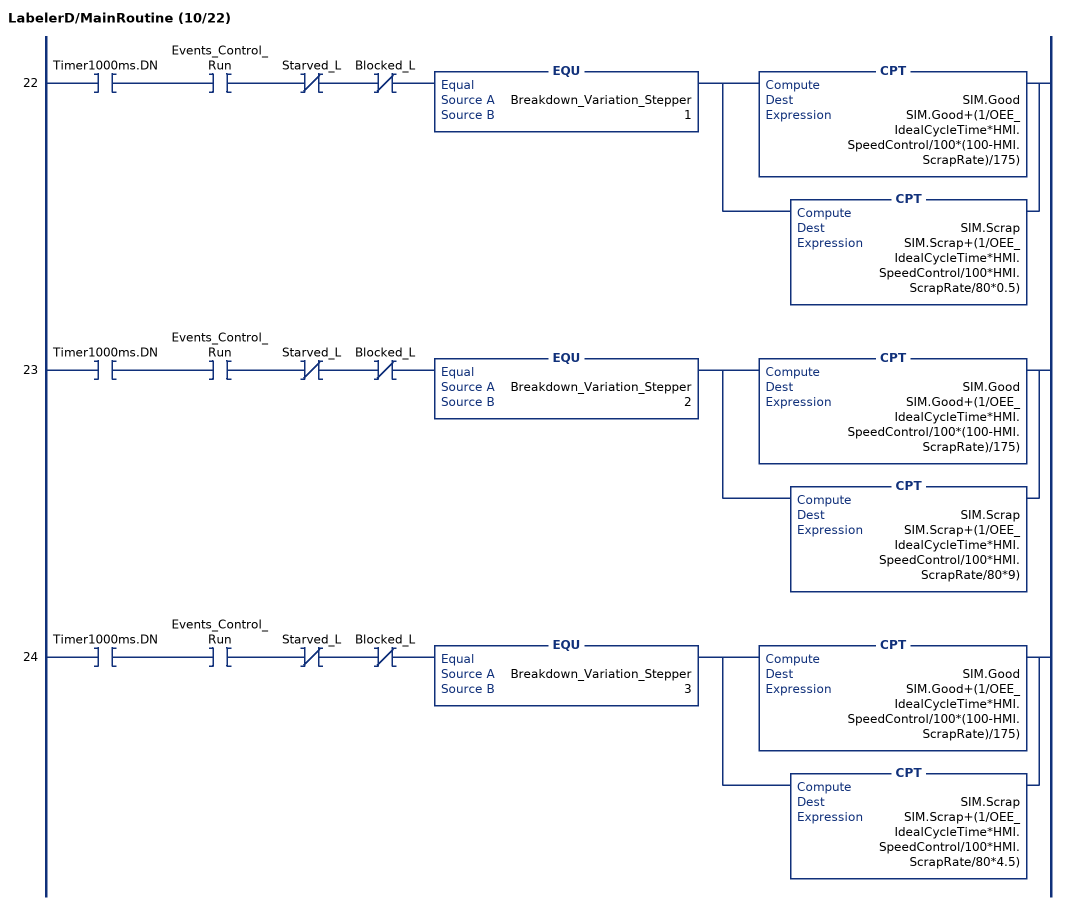
   22: XIC(Timer1000ms.DN)XIC(Events_Control_Run)XIO(Starved_L)XIO(Blocked_L)EQU(Breakdown_Variation_Stepper,1)[CPT(SIM.Good,SIM.Good+(1/OEE_IdealCycleTime*HMI.SpeedControl/100*(100-HMI.ScrapRate)/175)) ,CPT(SIM.Scrap,SIM.Scrap+(1/OEE_IdealCycleTime*HMI.SpeedControl/100*HMI.ScrapRate/80*0.5)) ];
   23: XIC(Timer1000ms.DN)XIC(Events_Control_Run)XIO(Starved_L)XIO(Blocked_L)EQU(Breakdown_Variation_Stepper,2)[CPT(SIM.Good,SIM.Good+(1/OEE_IdealCycleTime*HMI.SpeedControl/100*(100-HMI.ScrapRate)/175)) ,CPT(SIM.Scrap,SIM.Scrap+(1/OEE_IdealCycleTime*HMI.SpeedControl/100*HMI.ScrapRate/80*9)) ];
   24: XIC(Timer1000ms.DN)XIC(Events_Control_Run)XIO(Starved_L)XIO(Blocked_L)EQU(Breakdown_Variation_Stepper,3)[CPT(SIM.Good,SIM.Good+(1/OEE_IdealCycleTime*HMI.SpeedControl/100*(100-HMI.ScrapRate)/175)) ,CPT(SIM.Scrap,SIM.Scrap+(1/OEE_IdealCycleTime*HMI.SpeedControl/100*HMI.ScrapRate/80*4.5)) ];
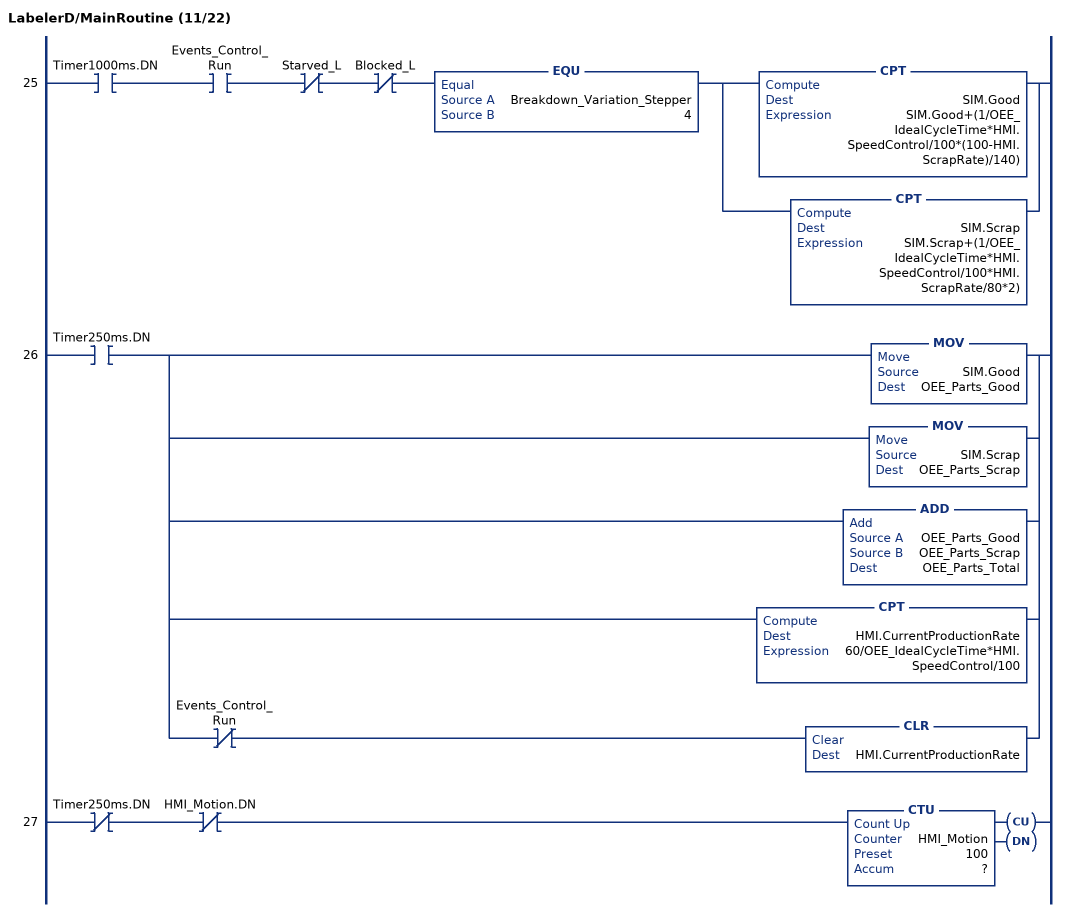
   25: XIC(Timer1000ms.DN)XIC(Events_Control_Run)XIO(Starved_L)XIO(Blocked_L)EQU(Breakdown_Variation_Stepper,4)[CPT(SIM.Good,SIM.Good+(1/OEE_IdealCycleTime*HMI.SpeedControl/100*(100-HMI.ScrapRate)/140)) ,CPT(SIM.Scrap,SIM.Scrap+(1/OEE_IdealCycleTime*HMI.SpeedControl/100*HMI.ScrapRate/80*2)) ];
   26: XIC(Timer250ms.DN)[[MOV(SIM.Good,OEE_Parts_Good) ,MOV(SIM.Scrap,OEE_Parts_Scrap) ,ADD(OEE_Parts_Good,OEE_Parts_Scrap,OEE_Parts_Total) ] ,CPT(HMI.CurrentProductionRate,60/OEE_IdealCycleTime*HMI.SpeedControl/100) ,XIO(Events_Control_Run) CLR(HMI.CurrentProductionRate) ];
   27: XIO(Timer250ms.DN)XIO(HMI_Motion.DN)CTU(HMI_Motion,?,?);
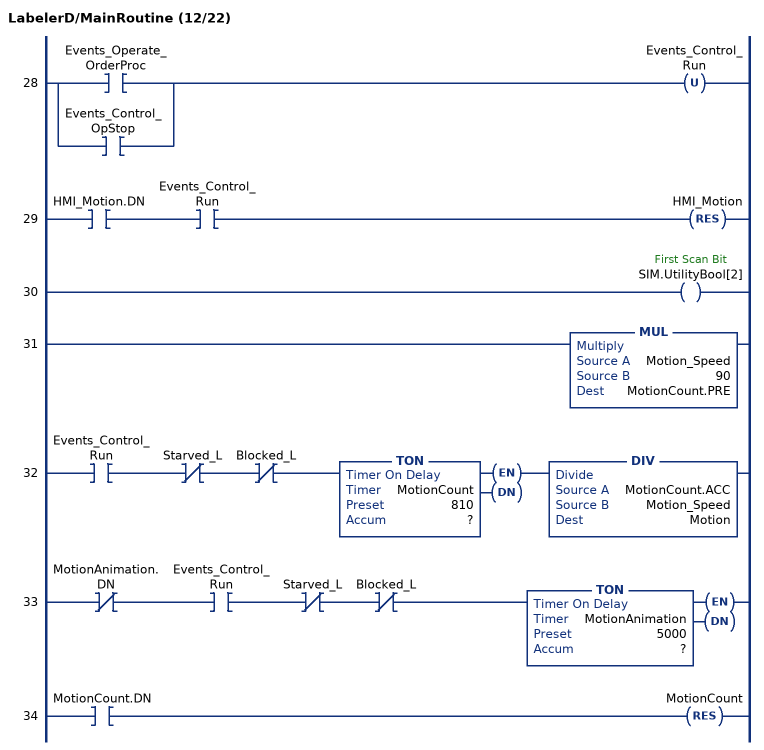
   28: [XIC(Events_Operate_OrderProc) ,XIC(Events_Control_OpStop) ]OTU(Events_Control_Run);
   29: XIC(HMI_Motion.DN)XIC(Events_Control_Run)RES(HMI_Motion);
   30: OTE(SIM.UtilityBool[2]);
   31: MUL(Motion_Speed,90,MotionCount.PRE);
   32: XIC(Events_Control_Run)XIO(Starved_L)XIO(Blocked_L)TON(MotionCount,?,?)DIV(MotionCount.ACC,Motion_Speed,Motion);
   33: XIO(MotionAnimation.DN)XIC(Events_Control_Run)XIO(Starved_L)XIO(Blocked_L)TON(MotionAnimation,?,?);
   34: XIC(MotionCount.DN)RES(MotionCount);
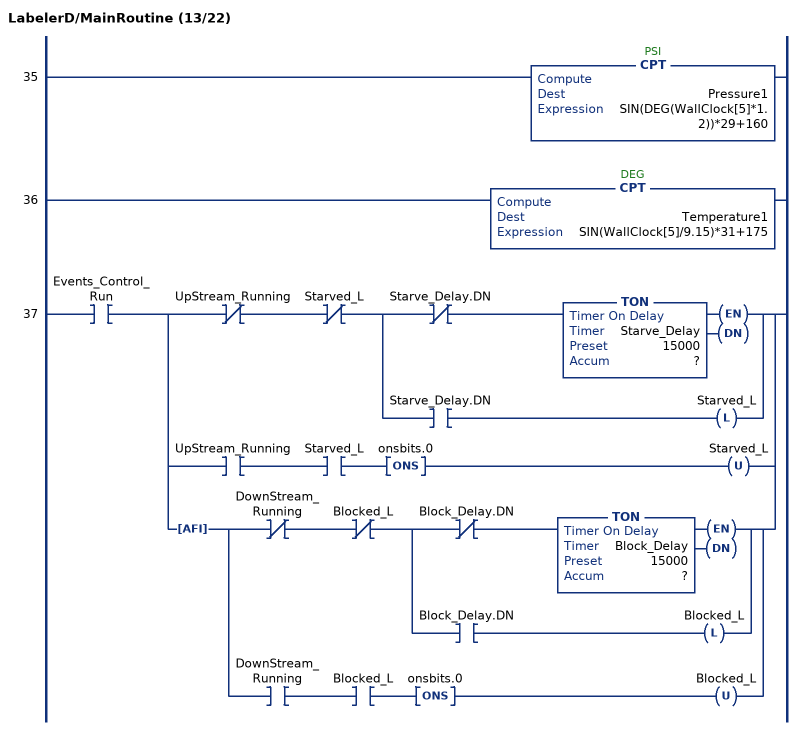
   35: CPT(Pressure1,SIN(DEG(WallClock[5]*1.2))*29+160);
   36: CPT(Temperature1,SIN(WallClock[5]/9.15)*31+175);
   37: XIC(Events_Control_Run)[[XIO(UpStream_Running) XIO(Starved_L) [XIO(Starve_Delay.DN) TON(Starve_Delay,?,?) ,XIC(Starve_Delay.DN) OTL(Starved_L) ] ,XIC(UpStream_Running) XIC(Starved_L) ONS(onsbits.0) OTU(Starved_L) ] ,AFI() [XIO(DownStream_Running) XIO(Blocked_L) [XIO(Block_Delay.DN) TON(Block_Delay,?,?) ,XIC(Block_Delay.DN) OTL(Blocked_L) ] ,XIC(DownStream_Running) XIC(Blocked_L) ONS(onsbits.0) OTU(Blocked_L) ] ];
